FUNCTION_BLOCK Merge_Split (* Composite Function Block Type *)
  (* Standard: 61499-2 *)
  (* Version 0.0, 9/22/2026, macie, Schneider Electric, template *)
  PACKAGE Main;
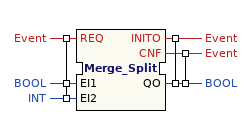
  EVENT_INPUT
    REQ WITH EI1, EI2; (* Normal Execution Request *)
  END_EVENT
  EVENT_OUTPUT
    INITO WITH QO; (* Initialization Confirm *)
    CNF WITH QO; (* Execution Confirmation *)
  END_EVENT
  VAR_INPUT
    EI1 : BOOL; (* Input event qualifier *)
    EI2 : INT;
  END_VAR
  VAR_OUTPUT
    QO : BOOL; (* Output event qualifier *)
  END_VAR
END_FUNCTION_BLOCK
